// TIA Portal V17 export
// export: Created 2025-03-05T08:00:46.7472738Z, ExportSetting WithDefaults, DisplayName Totally Integrated Automation Portal, DisplayVersion V17 Update 8, DisplayName TIA Portal Openness, DisplayVersion V17 Update 8, DisplayName TIA Portal Version Control Interface, DisplayVersion V17, DisplayName SINAMICS Startdrive Advanced, DisplayVersion V17 SP2, DisplayName SINAMICS Startdrive G110M, G120, G120C, G120D, G120P, G115D, DisplayVersion V17 SP2, DisplayName SINAMICS Startdrive G130, G150, S120, S150, SINAMICS MV, S210, DisplayVersion V17 SP2, DisplayName STEP 7 Professional, DisplayVersion V17 Update 8, DisplayName SINUMERIK ONE STEP 7 Toolbox, DisplayVersion V17 Update 12, DisplayName SINUMERIK 840D sl STEP 7 Toolbox, DisplayVersion V17 Update 12, DisplayName STEP 7 Safety, DisplayVersion V17 Update 6, DisplayName WinCC Advanced, DisplayVersion V17 Update 8
DATA_BLOCK "DB1101_MACHINE_SEQUENCE"   // DB1101
{ S7_Optimized_Access := 'FALSE'; DB_Accessible_From_OPC_UA := 'FALSE' }
AUTHOR : ETXETAR
VERSION : 1.0
// stored: AutoNumber false, DBAccessibleFromOPCUA false, DBAccessibleFromWebserver true, IsOnlyStoredInLoadMemory false, IsWriteProtectedInAS false
   VAR RETAIN
      GENERAL_CONDITIONS : Bool;   // MACHINING SEQUENCE GENERAL CONDITIONS / MACHINE SEQUENCE GENERAL CONDITIONS
      INITIAL_CONDITIONS : Bool;   // MACHINING SEQUENCE INITIAL CONDITIONS / MACHINE SEQUENCE INITIAL CONDITIONS
      START_REQUEST : Bool;   // MACHINING SEQUENCE START REQUEST / MACHINE SEQUENCE START REQUEST
      COMMAND : Bool;   // MACHINING SEQUENCE COMMAND / MACHINE SEQUENCE COMMAND
      REQUEST : Bool;   // MACHINING SEQUENCE REQUEST DELAYED / MACHINE SEQUENCE REQUEST
      COMMAND_PULSE : Bool;   // MACHINING SEQUENCE COMMAND PULSE / MACHINE SEQUENCE COMMAND PULSE
      REQUEST_PULSE : Bool;   // MACHINING SEQUENCE REQUEST PULSE / MACHINE SEQUENCE REQUEST PULSE
      RUNNING : Bool;   // MACHINING SEQUENCE IN PROCESS / MACHINE SEQUENCE RUNNING
      CYCLE_UNIT_01 : Bool;   // MACHINING SEQUENCE CYCLE STATION 01R / MACHINE SEQUENCE CYCLE UNIT 01
      CYCLE_UNIT_02 : Bool;   // MACHINING SEQUENCE CYCLE STATION 01L / MACHINE SEQUENCE CYCLE UNIT 02
      CYCLE_UNIT_03 : Bool;   // MACHINING SEQUENCE CYCLE STATION 01L / MACHINE SEQUENCE CYCLE UNIT 03
      NO_PART_AT_FEED_UNIT_01 : Bool;   // MACHINING SEQUENCE CYCLE STATION FIXTURE / MACHINE SEQUENCE NO PART AT FEED UNIT 02
      DELIVERY_OCCUPIED_UNIT_01 : Bool;   // MACHINING SEQUENCE CYCLE PART HANDLING DEVICE / MACHINE SEQUENCE DELIVERY OCCUPIED UNIT 02
      NO_PART_AT_FEED_UNIT_02 : Bool;   // MACHINING SEQUENCE NO PART AT FEED / MACHINE SEQUENCE NO PART AT FEED UNIT 02
      DELIVERY_OCCUPIED_UNIT_02 : Bool;   // MACHINING SEQUENCE DELIVERY OCCUPIED / MACHINE SEQUENCE DELIVERY OCCUPIED UNIT 02
      CLEAR_TO_LOAD_UNLOAD_UNIT_01 : Bool;   // MACHINING SEQUENCE OUT OF COLLISION TO PART HANDLING DEVICE / MACHINE SEQUENCE CLEAR TO LOAD UNLOAD MACHINE UNIT 01
      CLEAR_TO_LOAD_UNLOAD_UNIT_02 : Bool;   // MACHINING SEQUENCE OUT OF COLLISION TO PART HANDLING DEVICE / MACHINE SEQUENCE CLEAR TO LOAD UNLOAD MACHINE UNIT 02
      SKIP_FIXTURE_UNIT_01 : Bool;   // MACHINING SEQUENCE CLAMP FIXTURE 1 / MACHINE SEQUENCE SKIP FIXTURE UNIT 01
      SKIP_FIXTURE_UNIT_02 : Bool;   // MACHINING SEQUENCE CLAMP FIXTURE 2 / MACHINE SEQUENCE SKIP FIXTURE UNIT 02
      SPARE_1 : Bool;   // MACHINING SEQUENCE UNCLAMP FIXTURE 1 / MACHINE SEQUENCE
      SPARE_2 : Bool;   // MACHINING SEQUENCE UNCLAMP FIXTURE 2 / MACHINE SEQUENCE
      RESET_PLC_AND_CNC : Bool;   // MACHINING SEQUENCE RESET PLC AND CNC / MACHINE SEQUENCE RESET PLC AND CNC
      FULL_DEPTH : Bool;   // MACHINING SEQUENCE FULL DEPTH / MACHINE SEQUENCE FULL DEPTH
      TIME_EXCEEDED : Bool;   // MACHINING SEQUENCE TIME EXCEEDED / MACHINE SEQUENCE TIME EXCEEDED
      PREALARM : Bool;   // MACHINING SEQUENCE PREALARM / MACHINE SEQUENCE PREALARM
      LOADER_CHECK_PART_READY : Bool;   // MACHINING SEQUENCE LOADER CHECK PART READY / MACHINE SEQUENCE LOADER CHECK PART READY
      LOADER_RESET_CHECK_PART_READY : Bool;   // MACHINING SEQUENCE RST LOADER CHECK PART READY / MACHINE SEQUENCE LOADER RESET CHECK PART READY
      PREALARM_GONE : Bool;   // MACHINING SEQUENCE PREALARM GONE / MACHINE SEQUENCE PREALARM GONE
      AUX1 : Bool;   // MACHINING SEQUENCE AUX1 / MACHINE SEQUENCE AUX1
      AUX2 : Bool;   // MACHINING SEQUENCE AUX2 / MACHINE SEQUENCE AUX2
      AUX3 : Bool;   // MACHINING SEQUENCE AUX3 / MACHINE SEQUENCE AUX3
      START_GENERAL_COND_HELP : Bool;   // MACHINING SEQUENCE START GENERAL CONDITIONS HELP / MACHINE SEQUENCE START GENERAL COND HELP
      START_INITIAL_COND_HELP : Bool;   // MACHINING SEQUENCE START INITIAL CONDITIONS HELP / MACHINE SEQUENCE START INITIAL COND HELP
      TIMER_MACHINE_START_REQUEST : TON_TIME;   // MACHINE SEQUENCE START REQUEST TIMER
      "TIMER_TIME _EXCEEDED" : TON_TIME;   // MACHINE SEQUENCE TIME EXCEEDED TIMER
      TIMER_UNLOAD_UNIT_01_DELAY : TON_TIME;   // MACHINE SEQUENCE UNLOAD UNIT 01 DELAY TIMER
      TIMER_LOAD_UNIT_01_DELAY : TON_TIME;   // MACHINE SEQUENCE LOAD UNIT 01 DELAY TIMER
      TIMER_UNLOAD_UNIT_02_DELAY : TON_TIME;   // MACHINE SEQUENCE UNLOAD UNIT 02 DELAY TIMER
      TIMER_LOAD_UNIT_02_DELAY : TON_TIME;   // MACHINE SEQUENCE LOAD UNIT 02 DELAY TIMER
   END_VAR
BEGIN
   TIMER_MACHINE_START_REQUEST.PT := T#3s;
   "TIMER_TIME _EXCEEDED".PT := T#800s;
   TIMER_UNLOAD_UNIT_01_DELAY.PT := T#500ms;
   TIMER_LOAD_UNIT_01_DELAY.PT := T#1s;
   TIMER_UNLOAD_UNIT_02_DELAY.PT := T#500ms;
   TIMER_LOAD_UNIT_02_DELAY.PT := T#1s;
END_DATA_BLOCK
